INTERFACE I_SnappySetupConfigTestFrameWork

METHOD UseTestFramework : I_SnappySetupConfigBuild
VAR_INPUT
	itfTestFramework	: I_TestFrameWorkAdapter;
END_VAR
END_METHOD

METHOD WithoutTestFramework : I_SnappySetupConfigBuild
VAR_INPUT CONSTANT
	sTestSuiteName 	: T_MaxString;
	sTestName		: T_MaxString;
END_VAR
END_METHOD

END_INTERFACE

(* stored: Version 1.1.0.1, ProductVersion 3.1.4026.18
   Itf I_SnappySetupConfigTestFrameWork: Id {7d911619-4bba-4a11-8679-3e81ddc87c9b}
   Method UseTestFramework: Id {bb5fa30c-d772-4a55-9831-d8b435dda75b}
   Method WithoutTestFramework: Id {32f9c252-96d3-4a1a-8e3e-d93d2be176b4} *)
